DATA_BLOCK "PN-INPUT"
{ S7_Optimized_Access := 'FALSE' }
VERSION : 0.1
   STRUCT
      "00" : Byte;   // Заглушка--------------------------------------
      a1 : Byte;   // 1захват команды
      b1 : Byte;   // 1состояния
      c1 : Byte;   // 1ошибки
      d1 : Byte;   // 1UO
      e1 : Byte;   // 1DO_BYTE1 Текущий ряд, линия 1
      f1 : Byte;   // 1DO_BYTE2 Позиция в ряду, линия 1
      g1 : Byte;   // 1DO_BYTE3 Текущий ряд, линия 2
      h1 : Byte;   // 1DO_BYTE4 Позиция в ряду, линия 2
      i1 : Byte;   // 1DO_BYTE5 Моточасы1
      J1 : Byte;   // 1DO_BYTE6 Моточасы2
      K1 : DWord;
      P1 : Byte;   // 1RTK1--------------------------------------------------------
      a2 : Byte;   // 2захват команды
      b2 : Byte;   // 2состояния
      c2 : Byte;   // 2ошибки
      d2 : Byte;   // 2UO
      e2 : Byte;   // 2DO_BYTE1 Текущий ряд, линия 1
      f2 : Byte;   // 2DO_BYTE2 Позиция в ряду, линия 1
      g2 : Byte;   // 2DO_BYTE3 Текущий ряд, линия 2
      h2 : Byte;   // 2DO_BYTE4 Позиция в ряду, линия 2
      i2 : Byte;   // 2DO_BYTE5 Моточасы1
      J2 : Byte;   // 2DO_BYTE6 Моточасы2
      K2 : DWord;
      P2 : Byte;   // 2RTK2---------------------------------------------------------------
      a3 : Byte;   // 3захват команды
      b3 : Byte;   // 3состояния
      c3 : Byte;   // 3ошибки
      d3 : Byte;   // 3UO
      e3 : Byte;   // 3DO_BYTE1 Текущий ряд, линия 1
      f3 : Byte;   // 3DO_BYTE2 Позиция в ряду, линия 1
      g3 : Byte;   // 3DO_BYTE3 Текущий ряд, линия 2
      h3 : Byte;   // 3DO_BYTE4 Позиция в ряду, линия 2
      i3 : Byte;   // 3DO_BYTE5 Моточасы1
      J3 : Byte;   // 3DO_BYTE6 Моточасы2
      K3 : DWord;
      P3 : Byte;   // 3RTK3-------------------------------------------------------
      a4 : Byte;   // 4захват команды
      b4 : Byte;   // 4состояния
      c4 : Byte;   // 4ошибки
      d4 : Byte;   // 4UO
      e4 : Byte;   // 4DO_BYTE1 Текущий ряд, линия 1
      f4 : Byte;   // 4DO_BYTE2 Позиция в ряду, линия 1
      g4 : Byte;   // 4DO_BYTE3 Текущий ряд, линия 2
      h4 : Byte;   // 4DO_BYTE4 Позиция в ряду, линия 2
      i4 : Byte;   // 4DO_BYTE5 Моточасы1
      J4 : Byte;   // 4DO_BYTE6 Моточасы2
      K4 : DWord;
      P4 : Byte;   // 4RTK4--------------------------------------------------------
      a5 : Byte;   // заглушка четности
      c5 : DWord;   // FA1------------------------------------------------
      g5 : DWord;   // FA1
      FA1_1_ETA : Word;   // FA1_1_ETA
      FA1_1_BSpeed : Word;   // FA1_1_Speed
      b6 : DWord;   // FA2------------------------------------------------------
      c6 : DWord;   // FA2
      FA2_1_ETA : Word;   // FA2_1_ETA
      FA2_1_BSpeed : Word;   // FA2_1_Speed
      f6 : DWord;   // FA3------------------------------------------------
      g6 : DWord;   // FA3
      FA3_1_ETA : Word;   // FA3_1_ETA
      FA3_1_BSpeed : Word;   // FA3_1_Speed
      J6 : DWord;   // FA23------------------------------------------------------
      K6 : DWord;   // FA23
      FA23_1_ETA : Word;   // FA23_1_ETA
      FA23_1_BSpeed : Word;   // FA23_1_Speed
      c7 : DWord;   // FA24------------------------------------------------
      g7 : DWord;   // FA24
      FA24_1_ETA : Word;   // FA24_1_ETA
      FA24_1_BSpeed : Word;   // FA24_1_Speed
      b7 : DWord;   // FA4------------------------------------------------------
      c8 : DWord;   // FA4
      FA4_1_ETA : Word;   // FA4_1_ETA
      FA4_1_BSpeed : Word;   // FA4_1_Speed
      f7 : DWord;   // FA5------------------------------------------------
      g8 : DWord;   // FA5
      FA5_1_ETA : Word;   // FA5_1_ETA
      FA5_1_BSpeed : Word;   // FA5_1_Speed
      J7 : DWord;   // FA20------------------------------------------------------
      K8 : DWord;   // FA20
      FA20_1_ETA : Word;   // FA20_1_ETA
      FA20_1_BSpeed : Word;   // FA20_1_Speed
      c9 : DWord;   // FA25_1------------------------------------------------
      g9 : DWord;   // FA25_1
      FA25_1_ETA : Word;   // FA25_1_ETA
      FA25_1_BSpeed : Word;   // FA25_1_Speed
      b8 : DWord;   // FA25_2------------------------------------------------------
      c10 : DWord;   // FA25_2
      FA25_2_ETA : Word;   // FA25_2_ETA
      FA25_2_BSpeed : Word;   // FA25_2_Speed
      f8 : DWord;   // FA6------------------------------------------------
      g10 : DWord;   // FA6
      FA6_1_ETA : Word;   // FA6_1_ETA
      FA6_1_BSpeed : Word;   // FA6_1_Speed
      J8 : DWord;   // FA7------------------------------------------------------
      K10 : DWord;   // FA7
      FA7_1_ETA : Word;   // FA7_1_ETA
      FA7_1_BSpeed : Word;   // FA7_1_Speed
      c11 : DWord;   // FA8------------------------------------------------
      g11 : DWord;   // FA8
      FA8_1_ETA : Word;   // FA8_1_ETA
      FA8_1_BSpeed : Word;   // FA8_1_Speed
      b9 : DWord;   // FA26------------------------------------------------------
      c12 : DWord;   // FA26
      FA26_1_ETA : Word;   // FA26_1_ETA
      FA26_1_BSpeed : Word;   // FA26_1_Speed
      f9 : DWord;   // FA27------------------------------------------------
      g12 : DWord;   // FA27
      FA27_1_ETA : Word;   // FA27_1_ETA
      FA27_1_BSpeed : Word;   // FA27_1_Speed
      J9 : DWord;   // FA9------------------------------------------------------
      K12 : DWord;   // FA9
      FA9_1_ETA : Word;   // FA9_1_ETA
      FA9_1_BSpeed : Word;   // FA9_1_Speed
      J10 : DWord;   // FA10------------------------------------------------------
      K13 : DWord;   // FA10
      FA10_1_ETA : Word;   // FA10_1_ETA
      FA10_1_BSpeed : Word;   // FA10_1_Speed
      f10 : DWord;   // FA28------------------------------------------------
      g13 : DWord;   // FA28
      FA28_1_ETA : Word;   // FA28_1_ETA
      FA28_1_BSpeed : Word;   // FA28_1_Speed
      N5 : Word;
      O5 : Word;
      temp : DWord;
      temp1 : DWord;
      temp2 : DWord;
   END_STRUCT;


BEGIN

END_DATA_BLOCK

